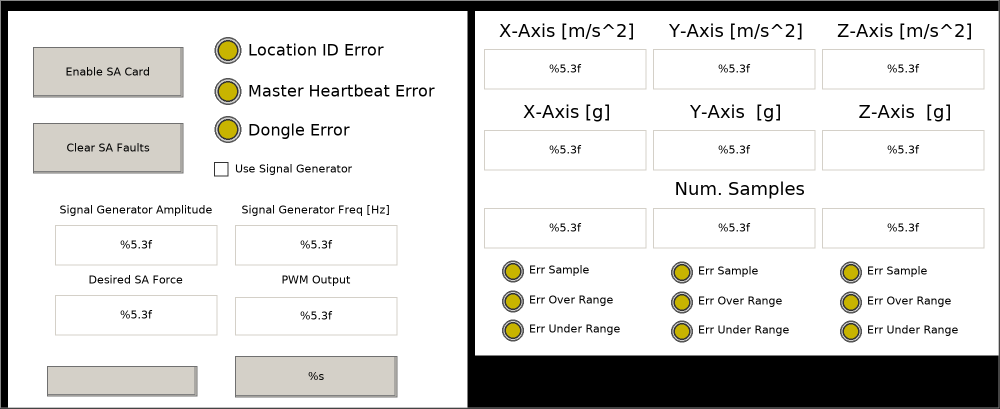
VISUALIZATION Visualization  // 1000x409
    RoundedRectangle (7,10 461x399)
    RoundedRectangle (474,10 526x346)
    Lamp1 (212,76 32x31), variable: MAIN.saErrMasterHb, style: Lamp-Lamp1-Yellow
    Lamp1 (212,114 32x31), variable: MAIN.saErrDongle, style: Lamp-Lamp1-Yellow
    Label (245,76 213x30), "Master Heartbeat Error"
    Label (245,115 213x30), "Dongle Error"
    Button (33,47 150x50), "Enable SA Card"
        toggle MAIN.saEnable
    Textfield (55,295 162x40), "%5.3f", text variable: MAIN.saForceSetting
        OnMouseClick: write MAIN.saForceSetting via Default
    Label (61,265 150x30), "Desired SA Force"
    Button (33,123 150x50), "Clear SA Faults"
        tap MAIN.saClearFault
    Textfield (235,297 162x38), "%5.3f", text variable: MAIN.saPwm1
    Label (241,265 150x30), "PWM Output"
    Label (492,97 150x30), "X-Axis [g]"
    Textfield (484,130 162x40), "%5.3f", text variable: MAIN.xAxisConverted_g
    Label (661,97 150x30), "Y-Axis [g]"
    Textfield (653,130 162x40), "%5.3f", text variable: MAIN.yAxisConverted_g
    Label (830,97 150x30), "Z-Axis [g]"
    Textfield (822,130 162x40), "%5.3f", text variable: MAIN.zAxisConverted_g
    Label (665,174 150x30), "Num. Samples"
    Textfield (484,208 162x40), "%5.3f", text variable: MAIN.xAxisNumSamples
    Textfield (653,208 162x40), "%5.3f", text variable: MAIN.yAxisNumSamples
    Textfield (822,208 162x40), "%5.3f", text variable: MAIN.ZAxisNumSamples
    Label (526,255 124x30), "Err Sample"
    Lamp1 (496,259 34x25), variable: MAIN.errXAxisSample, style: Lamp-Lamp1-Yellow
    Label (526,285 124x30), "Err Over Range"
    Lamp1 (496,289 34x25), variable: MAIN.errXAxisOverRnge, style: Lamp-Lamp1-Yellow
    Label (526,314 124x30), "Err Under Range"
    Lamp1 (496,318 34x25), variable: MAIN.errXAxisUndrRnge, style: Lamp-Lamp1-Yellow
    Label (695,256 124x30), "Err Sample"
    Lamp1 (665,260 34x25), variable: MAIN.errYAxisSample, style: Lamp-Lamp1-Yellow
    Label (695,286 124x30), "Err Over Range"
    Lamp1 (665,290 34x25), variable: MAIN.errYAxisOverRnge, style: Lamp-Lamp1-Yellow
    Label (695,315 124x30), "Err Under Range"
    Lamp1 (665,319 34x25), variable: MAIN.errYAxisUndrRnge, style: Lamp-Lamp1-Yellow
    Label (864,256 124x30), "Err Sample"
    Lamp1 (834,260 34x25), variable: MAIN.errZAxisSample, style: Lamp-Lamp1-Yellow
    Label (864,286 124x30), "Err Over Range"
    Lamp1 (834,290 34x25), variable: MAIN.errZAxisOverRnge, style: Lamp-Lamp1-Yellow
    Label (864,315 124x30), "Err Under Range"
    Lamp1 (834,319 34x25), variable: MAIN.errYAxisUndrRnge, style: Lamp-Lamp1-Yellow
    Button (235,356 162x41), "%s", text variable: MAIN.sPyTestMsg
        toggle MAIN.tglPyTest
    Lamp1 (212,35 32x31), variable: MAIN.saErrLocId, style: Lamp-Lamp1-Yellow
    Label (245,35 213x30), "Location ID Error"
    Checkbox (212,154 234x30), "Use Signal Generator", variable: MAIN.bUseSigGen
    Label (241,195 150x30), "Signal Generator Freq [Hz]"
    Textfield (235,225 162x40), "%5.3f", text variable: MAIN.sigGenFreq
        OnMouseClick: write MAIN.sigGenFreq via Default
    Label (492,16 150x30), "X-Axis [m/s^2]"
    Textfield (484,49 162x40), "%5.3f", text variable: MAIN.xAxisConverted_mps2
    Label (661,16 150x30), "Y-Axis [m/s^2]"
    Textfield (653,49 162x40), "%5.3f", text variable: MAIN.yAxisConverted_mps2
    Label (830,16 150x30), "Z-Axis [m/s^2]"
    Textfield (822,49 162x40), "%5.3f", text variable: MAIN.zAxisConverted_mps2
    Label (61,195 150x30), "Signal Generator Amplitude"
    Textfield (55,225 162x40), "%5.3f", text variable: MAIN.stCTRL_SIGNAL_GENERATOR_PARAMS.fAmplitude
        OnMouseClick: write MAIN.stCTRL_SIGNAL_GENERATOR_PARAMS.fAmplitude via Default
    Button (47,366 150x30)
        toggle MAIN.test
END_VISUALIZATION

(* stored: Version 1.1.0.1
   Visu Visualization: Id {4066fa24-1414-4763-8661-51269ac20cff} *)
